// TwinCAT 3 PLC project UnitTestLib
// Title: Unittest
// Company: Hoox.Software
// Author: Patrick Dressel
// ProjectVersion: 0.1
// Description: Basisfunktion zur Erstellung von Unittest und Dokumentation.
// ProgramVersion: 3.1.4022.2
// libraries:
//   Tc2_Standard, * (Beckhoff Automation GmbH)
//   Tc2_System, * (Beckhoff Automation GmbH)
//   Tc2_Utilities, * (Beckhoff Automation GmbH)
//   Base Interfaces,newest,System
// project tree:
//   Datatypes/ EResult_t.TcDUT, EState_t.TcDUT, ObjectId_t.TcDUT (not stored), SResult_t.TcDUT (not stored), SStatistic_t.TcDUT (not stored), StringHandle_t.TcDUT, IdHandle_t.TcDUT, StrMessage_t.TcDUT (not stored), TestCaseHandle_t.TcDUT, TestSuiteHandle_t.TcDUT (not stored)
//   Datatypes/Report/ EExportState_t.TcDUT (not stored), ERetCode_t.TcDUT, NameHandle_t.TcDUT, PathHandle_t.TcDUT, StrFileName_t.TcDUT (not stored), StrPathName_t.TcDUT, UBaseTypes_t.TcDUT (not stored), UTime_t.TcDUT (not stored)
//   Source/ FB_Testsuite.TcPOU, FB_UnitTestBase.TcPOU, PRG_UnitTestLib.TcPOU
//   Source/Report/ FB_TestReportBase.TcPOU, FB_TextReport.TcPOU
//   Version/ Global_Version.TcGVL

// ---- Datatypes/EResult_t.TcDUT
{attribute 'qualified_only'}
{attribute 'strict'}
TYPE EResult_t :
(
	eStatePassed,
	eStateFailed,
	eStateFailedFatal
);
END_TYPE

// ---- Datatypes/EState_t.TcDUT
{attribute 'qualified_only'}
{attribute 'strict'}
TYPE EState_t :
(
	eStateInit,
	eStateIdle,
	eStatePrepare,
	eStateExecute,
	eStateCleanUp,
	eStateReady,
	eStateError
);
END_TYPE

// ---- Datatypes/Report/ERetCode_t.TcDUT
{attribute 'qualified_only'}
{attribute 'strict'}
TYPE ERetCode_t :
(
	eRetFailed := 0,
	eRetBusy,
	eRetDone
);
END_TYPE

// ---- Datatypes/Report/NameHandle_t.TcDUT
TYPE NameHandle_t : Pointer to StrFileName_t; END_TYPE

// ---- Datatypes/Report/PathHandle_t.TcDUT
TYPE PathHandle_t : Pointer to StrFileName_t; END_TYPE

// ---- Datatypes/Report/StrPathName_t.TcDUT
TYPE StrPathName_t : String(255); END_TYPE

// ---- Datatypes/StringHandle_t.TcDUT
TYPE StringHandle_t : POINTER TO STRING(255); END_TYPE

// ---- Datatypes/IdHandle_t.TcDUT
TYPE IdHandle_t : POINTER TO ObjectId_t; END_TYPE

// ---- Datatypes/TestCaseHandle_t.TcDUT
TYPE TestCaseHandle_t : POINTER TO FB_UnitTestBase; END_TYPE

// ---- Version/Global_Version.TcGVL
{attribute 'TcGenerated'}
// This function has been automatically generated from the project information.
VAR_GLOBAL CONSTANT
	{attribute 'const_non_replaced'}
	{attribute 'linkalways'}
	stLibVersion_Unittest : ST_LibVersion := (iMajor := 0, iMinor := 1, iBuild := 0, iRevision := 0, sVersion := '0.1');
END_VAR

// ---- Source/FB_Testsuite.TcPOU
(******************************************************************************
Baustein: FB_Testsuite
Spezifikation: doc/Spezifikation.pdf, Kap. x.y.z
-------------------------------------------------------------------------------
erstellt:
von:
Geändert:
von:
-------------------------------------------------------------------------------
Beschreibung
Dieser Baustein enthält alle zugeordneten Testfälle. Ein Testfall
ist ein abgeleiteter Baustein (FB) von FB_UnitTestBase.

-------------------------------------------------------------------------------
Input
-

Output
-
******************************************************************************)
FUNCTION_BLOCK FB_Testsuite
VAR_INPUT
	i_bStart : BOOL;
END_VAR
VAR_OUTPUT
	o_eState  		: EState_t;
	o_eResult 		: EResult_t;
END_VAR
VAR
	strId			: ObjectId_t;
	bRegistered     : BOOL;
	a_pTest  		: ARRAY [0..255] OF TestCaseHandle_t;
	pTest     		: TestCaseHandle_t;
	u16TestCases  	: UINT;
	u16Index 		: UINT;
	sStatistic 		: SStatistic_t;
END_VAR


	CASE o_eState OF
		
	EState_t.eStateInit:
	
		o_eState 	:= EState_t.eStateError;
		IF bRegistered = TRUE THEN
			o_eState 	:= EState_t.eStateIdle;
		END_IF;
		
	EState_t.eStateIdle:

		u16Index := 0;

		IF i_bStart = TRUE THEN
			logInfo(CONCAT('Run Testsuite ', strId));
			pTest 	 := getFirstTestCase();
			o_eState  := EState_t.eStatePrepare;
			o_eResult := EResult_t.eStatePassed;
		END_IF;

	EState_t.eStatePrepare:
	
		sStatistic.u32Executed  := 0;
		sStatistic.u32Passed 	:= 0;
		sStatistic.u32Failed 	:= 0;
		sStatistic.u32Asserts 	:= 0;

		IF pTest <> 0 THEN
			IF pTest^.prepare() = TRUE THEN
				pTest 	:= getNextTestCase();
			END_IF;
		ELSE
			o_eState := EState_t.eStateExecute;
			pTest 	:= getFirstTestCase();
		END_IF;

	EState_t.eStateExecute:

		IF pTest <> 0 THEN
			IF pTest^.execute() = TRUE THEN

				sStatistic.u32Executed := sStatistic.u32Executed + 1;	
			
				sStatistic.u32Passed 	:= sStatistic.u32Passed + pTest^.getPassed();
				sStatistic.u32Failed 	:= sStatistic.u32Failed + pTest^.getFailed();
				sStatistic.u32Asserts   := sStatistic.u32Passed + sStatistic.u32Failed;
				
				CASE o_eResult OF 

				EResult_t.eStatePassed:
					// Status des letzen Tests übernehmen
					o_eResult := pTest^.o_eResult;

				EResult_t.eStateFailed:
					// Status nur übernehmen wenn ein Fatal-Status
					// ermittelt wird und der Test sofort abgebrochen
					// werden soll.
					IF pTest^.o_eResult = EResult_t.eStateFailedFatal THEN
						o_eResult := pTest^.o_eResult;
						o_eState  := EState_t.eStateCleanUp;
						pTest 	  := getFirstTestCase();	
					END_IF;

				EResult_t.eStateFailedFatal:

					o_eState := EState_t.eStateCleanUp;
					pTest 	:= getFirstTestCase();					

				END_CASE;

				IF o_eResult <> EResult_t.eStateFailedFatal THEN
					pTest 	 := getNextTestCase();
				END_IF;

			END_IF;
		ELSE
			o_eState := EState_t.eStateCleanUp;
			pTest 	:= getFirstTestCase();
		END_IF;

	ESTate_t.eStateCleanUp:

		IF pTest <> 0 THEN
			IF pTest^.cleanup() = TRUE THEN
				pTest 	:= getNextTestCase();
			END_IF;
		ELSE
			o_eState := EState_t.eStateReady;
		END_IF;
		
	ESTate_t.eStateReady:
	
		IF i_bStart = FALSE THEN
			o_eState := EState_t.eStateIdle;
		END_IF
		
	ESTate_t.eStateError:	
		
		// wenn wir hier rauskommen ist was dummes passiert
		
	ELSE
		
		o_eState := EState_t.eStateError;
		
	END_CASE;
	
	
	
	
	
	
//

(******************************************************************************
Baustein: FB_UnitTestBase.
Spezifikation: doc/Spezifikation.pdf, Kap. x.y.z
-------------------------------------------------------------------------------
erstellt:
von:
Geändert:
von:
-------------------------------------------------------------------------------
Beschreibung
Diese Methode

-------------------------------------------------------------------------------
Input
-

Output
-
******************************************************************************)
METHOD PUBLIC addTestcase : BOOL
VAR_INPUT
	i_pTestCase : TestCaseHandle_t;
END_VAR

	addTestcase := FALSE;

	IF 	i_pTestCase  <> 0   AND 
		u16TestCases <  255 THEN
		
		a_pTest[u16TestCases] := i_pTestCase;
		
		u16TestCases := u16TestCases +1;
		
		sStatistic.u32TestCases := sStatistic.u32TestCases + 1;
		
		addTestcase := true;
	END_IF
END_METHOD

METHOD FB_init : BOOL
VAR_INPUT
	bInitRetains 	: BOOL; // if TRUE, the retain variables are initialized (warm start / cold start)
	bInCopyCode 	: BOOL;  // if TRUE, the instance afterwards gets moved into the copy code (online change)
	i_strId	  		: ObjectId_t;
END_VAR

	strId := i_StrId;
	
	register();
END_METHOD

METHOD PUBLIC getExecuted : UDINT
VAR_INPUT
END_VAR

	getExecuted := sStatistic.u32Executed;
END_METHOD

METHOD PUBLIC getFailed : UDINT
VAR_INPUT
END_VAR

	getFailed := sStatistic.u32Failed;
END_METHOD

(******************************************************************************
Baustein: FB_UnitTestBase.
Spezifikation: doc/Spezifikation.pdf, Kap. x.y.z
-------------------------------------------------------------------------------
erstellt:
von:
Geändert:
von:
-------------------------------------------------------------------------------
Beschreibung
Diese Methode

-------------------------------------------------------------------------------
Input
-

Output
-
******************************************************************************)
METHOD PRIVATE getFirstTestCase : TestCaseHandle_t
VAR_INPUT
END_VAR

	u16Index := 0;
	getFirstTestCase := a_pTest[0];
END_METHOD

METHOD PUBLIC getId : STRING
VAR_INPUT
END_VAR

	getId := strId;
END_METHOD

(******************************************************************************
Baustein: FB_UnitTestBase.
Spezifikation: doc/Spezifikation.pdf, Kap. x.y.z
-------------------------------------------------------------------------------
erstellt:
von:
Geändert:
von:
-------------------------------------------------------------------------------
Beschreibung
Diese Methode

-------------------------------------------------------------------------------
Input
-

Output
-
******************************************************************************)
METHOD PRIVATE getNextTestCase : TestCaseHandle_t
VAR_INPUT
END_VAR

	getNextTestCase := 0;
	u16Index 		 := u16Index + 1;

	IF u16Index < u16TestCases THEN
		getNextTestCase := a_pTest[u16Index];
	END_IF;
END_METHOD

METHOD PUBLIC getNoOfAsserts : UDINT
VAR_INPUT
END_VAR

	getNoOfAsserts := sStatistic.u32Asserts;
END_METHOD

METHOD PUBLIC getNoOfTests : UDINT
VAR_INPUT
END_VAR

	getNoOfTests := sStatistic.u32TestCases;
END_METHOD

METHOD PUBLIC getPassed : UDINT
VAR_INPUT
END_VAR

	getPassed := sStatistic.u32Passed;
END_METHOD

METHOD PROTECTED logInfo : BOOL
VAR_INPUT
	i_strMessage : StrMessage_t;
END_VAR

	ADSLOGSTR(msgCtrlMask 	:= ADSLOG_MSGTYPE_HINT , 
			  msgFmtStr 	:= i_strMessage, 
			  strArg 		:= '');
END_METHOD

(******************************************************************************
Baustein: FB_UnitTestBase.
Spezifikation: doc/Spezifikation.pdf, Kap. x.y.z
-------------------------------------------------------------------------------
erstellt:
von:
Geändert:
von:
-------------------------------------------------------------------------------
Beschreibung
Diese Methode

-------------------------------------------------------------------------------
Input
-

Output
-
******************************************************************************)
METHOD PROTECTED register : BOOL
VAR_INPUT
END_VAR

	bRegistered := PRG_UnitTestLib.addTestSuite(this);
END_METHOD

END_FUNCTION_BLOCK

// ---- Source/FB_UnitTestBase.TcPOU
(******************************************************************************
Baustein: FB_UnitTestBase
Spezifikation: doc/Spezifikation.pdf, Kap. x.y.z
-------------------------------------------------------------------------------
erstellt:
von:
Geändert:
von:
-------------------------------------------------------------------------------
Beschreibung
Dieser Baustein stellt die Basis für einen Unittest dar und enthält
alle notwendigen Variablen und Methoden zur Testauswertung.

-------------------------------------------------------------------------------
Input
-

Output
-
******************************************************************************)
FUNCTION_BLOCK FB_UnitTestBase
VAR_INPUT
END_VAR
VAR_OUTPUT
	o_eState : EState_t;
	o_eResult: EResult_t;
END_VAR
VAR
	strId	  		: ObjectId_t;
	pTestSuite      : TestSuiteHandle_t;
	bRegistered 	: BOOL;
	u32Passed 		: UDINT;
	u32Failed 		: UDINT;
END_VAR

(******************************************************************************
Baustein: FB_UnitTestBase.addFailed
Spezifikation: doc/Spezifikation.pdf, Kap. x.y.z
-------------------------------------------------------------------------------
erstellt:
von:
Geändert:
von:
-------------------------------------------------------------------------------
Beschreibung
Diese Methode

-------------------------------------------------------------------------------
Input
-

Output
-
******************************************************************************)
METHOD PRIVATE addFailed : BOOL
VAR_INPUT
	bFatal : BOOL;
END_VAR

	u32Failed := u32Failed + 1;
	
	o_eResult := EResult_t.eStateFailed;
	
	IF bFatal = true THEN
		o_eResult := EResult_t.eStateFailedFatal;
		logError(concat('Test Failed Fatal: ', strId));
	ELSE
		logError(concat('Test Failed : ', strId));
	END_IF
END_METHOD

(******************************************************************************
Baustein: FB_UnitTestBase.
Spezifikation: doc/Spezifikation.pdf, Kap. x.y.z
-------------------------------------------------------------------------------
erstellt:
von:
Geändert:
von:
-------------------------------------------------------------------------------
Beschreibung
Diese Methode

-------------------------------------------------------------------------------
Input
-

Output
-
******************************************************************************)
METHOD PRIVATE addPassed : BOOL
VAR_INPUT
END_VAR

	u32Passed := u32Passed + 1;
END_METHOD

METHOD PROTECTED assertEQUAL : BOOL
VAR_INPUT
	Actual   : ANY;
	Expected : ANY;
END_VAR

	assertEQUAL := FALSE;
	
	IF validate(Actual, Expected) = FALSE THEN
		addFailed(true);
		RETURN;
	END_IF
	
	assertTrue(MEMCMP(Actual.pValue, Expected.pValue, TO_UDINT(Actual.diSize)) = 0);
END_METHOD

METHOD PROTECTED assertEQUAL_Fatal : BOOL
VAR_INPUT
	Actual   : ANY;
	Expected : ANY;
END_VAR

	assertEQUAL_Fatal := FALSE;
	
	IF validate(Actual, Expected) = FALSE THEN
		addFailed(true);
		RETURN;
	END_IF

	assertTrue_Fatal(MEMCMP(Actual.pValue, Expected.pValue, TO_UDINT(Actual.diSize)) = 0);
END_METHOD

(******************************************************************************
Baustein: FB_UnitTestBase.assertFALSE
Spezifikation: doc/Spezifikation.pdf, Kap. x.y.z
-------------------------------------------------------------------------------
erstellt:
von:
Geändert:
von:
-------------------------------------------------------------------------------
Beschreibung
Diese Methode...

-------------------------------------------------------------------------------
Input
-

Output
-
******************************************************************************)
METHOD PROTECTED assertFALSE : BOOL
VAR_INPUT
	bValue : BOOL;
END_VAR

	IF bValue = FALSE THEN
		u32Passed := u32Passed + 1;
	ELSE
		u32Failed := u32Failed + 1;
	END_IF
END_METHOD

(******************************************************************************
Baustein: FB_UnitTestBase.
Spezifikation: doc/Spezifikation.pdf, Kap. x.y.z
-------------------------------------------------------------------------------
erstellt:
von:
Geändert:
von:
-------------------------------------------------------------------------------
Beschreibung
Diese Methode

-------------------------------------------------------------------------------
Input
-

Output
-
******************************************************************************)
METHOD PROTECTED assertFALSE_Fatal : BOOL
VAR_INPUT
	bValue : BOOL;
END_VAR

	IF bValue = FALSE THEN
		addPassed();
	ELSE
		addFailed(bFatal := true);
	END_IF
END_METHOD

METHOD PROTECTED assertNotEqual : BOOL
VAR_INPUT
	Actual   : ANY;
	Expected : ANY;
END_VAR

	assertNotEqual := FALSE;
	
	IF validate(Actual, Expected) = FALSE THEN
		addFailed(true);
		RETURN;
	END_IF
	
	assertTrue(MEMCMP(Actual.pValue, Expected.pValue, TO_UDINT(Actual.diSize)) <> 0);
END_METHOD

METHOD PROTECTED assertNotEqual_Fatal : BOOL
VAR_INPUT
	Actual   : ANY;
	Expected : ANY;
END_VAR

	assertNotEqual_Fatal := FALSE;
	
	IF validate(Actual, Expected) = FALSE THEN
		addFailed(true);
		RETURN;
	END_IF
	
	assertTrue_Fatal(MEMCMP(Actual.pValue, Expected.pValue, TO_UDINT(Actual.diSize)) <> 0);
END_METHOD

(******************************************************************************
Baustein: FB_UnitTestBase.
Spezifikation: doc/Spezifikation.pdf, Kap. x.y.z
-------------------------------------------------------------------------------
erstellt:
von:
Geändert:
von:
-------------------------------------------------------------------------------
Beschreibung
Diese Methode

-------------------------------------------------------------------------------
Input
-

Output
-
******************************************************************************)
METHOD PROTECTED assertPtrEqual : BOOL
VAR_INPUT
	pActual   : PVOID;
	pExpected : PVOID;
END_VAR

	assertTRUE(pActual = pExpected);
END_METHOD

(******************************************************************************
Baustein: FB_UnitTestBase.
Spezifikation: doc/Spezifikation.pdf, Kap. x.y.z
-------------------------------------------------------------------------------
erstellt:
von:
Geändert:
von:
-------------------------------------------------------------------------------
Beschreibung
Diese Methode

-------------------------------------------------------------------------------
Input
-

Output
-
******************************************************************************)
METHOD PROTECTED assertPtrEqual_Fatal : BOOL
VAR_INPUT
	pActual   : PVOID;
	pExpected : PVOID;
END_VAR

	assertTRUE_Fatal(pActual = pExpected);
END_METHOD

(******************************************************************************
Baustein: FB_UnitTestBase.
Spezifikation: doc/Spezifikation.pdf, Kap. x.y.z
-------------------------------------------------------------------------------
erstellt:
von:
Geändert:
von:
-------------------------------------------------------------------------------
Beschreibung
Diese Methode

-------------------------------------------------------------------------------
Input
-

Output
-
******************************************************************************)
METHOD PROTECTED assertPtrNotEqual : BOOL
VAR_INPUT
	pActual   : PVOID;
	pExpected : PVOID;
END_VAR

	assertTRUE(pActual <> pExpected);
END_METHOD

(******************************************************************************
Baustein: FB_UnitTestBase.
Spezifikation: doc/Spezifikation.pdf, Kap. x.y.z
-------------------------------------------------------------------------------
erstellt:
von:
Geändert:
von:
-------------------------------------------------------------------------------
Beschreibung
Diese Methode

-------------------------------------------------------------------------------
Input
-

Output
-
******************************************************************************)
METHOD PROTECTED assertPtrNotEqual_Fatal : BOOL
VAR_INPUT
	pActual   : PVOID;
	pExpected : PVOID;
END_VAR

	assertTRUE_Fatal(pActual <> pExpected);
END_METHOD

(******************************************************************************
Baustein: FB_UnitTestBase.
Spezifikation: doc/Spezifikation.pdf, Kap. x.y.z
-------------------------------------------------------------------------------
erstellt:
von:
Geändert:
von:
-------------------------------------------------------------------------------
Beschreibung
Diese Methode

-------------------------------------------------------------------------------
Input
-

Output
-
******************************************************************************)
METHOD PROTECTED assertPtrNotNull : BOOL
VAR_INPUT
	pActual   : PVOID;
END_VAR

	assertTRUE(pActual <> 0);
END_METHOD

(******************************************************************************
Baustein: FB_UnitTestBase.
Spezifikation: doc/Spezifikation.pdf, Kap. x.y.z
-------------------------------------------------------------------------------
erstellt:
von:
Geändert:
von:
-------------------------------------------------------------------------------
Beschreibung
Diese Methode

-------------------------------------------------------------------------------
Input
-

Output
-
******************************************************************************)
METHOD PROTECTED assertPtrNotNull_Fatal : BOOL
VAR_INPUT
	pActual   : PVOID;
END_VAR

	assertTRUE_Fatal(pActual <> 0);
END_METHOD

(******************************************************************************
Baustein: FB_UnitTestBase.
Spezifikation: doc/Spezifikation.pdf, Kap. x.y.z
-------------------------------------------------------------------------------
erstellt:
von:
Geändert:
von:
-------------------------------------------------------------------------------
Beschreibung
Diese Methode

-------------------------------------------------------------------------------
Input
-

Output
-
******************************************************************************)
METHOD PROTECTED assertPtrNull : BOOL
VAR_INPUT
	pActual   : PVOID;
END_VAR

	assertTRUE(pActual = 0);
END_METHOD

(******************************************************************************
Baustein: FB_UnitTestBase.
Spezifikation: doc/Spezifikation.pdf, Kap. x.y.z
-------------------------------------------------------------------------------
erstellt:
von:
Geändert:
von:
-------------------------------------------------------------------------------
Beschreibung
Diese Methode

-------------------------------------------------------------------------------
Input
-

Output
-
******************************************************************************)
METHOD PROTECTED assertPtrNull_Fatal : BOOL
VAR_INPUT
	pActual   : PVOID;
END_VAR

	assertTRUE_Fatal(pActual = 0);
END_METHOD

(******************************************************************************
Baustein: FB_UnitTestBase.
Spezifikation: doc/Spezifikation.pdf, Kap. x.y.z
-------------------------------------------------------------------------------
erstellt:
von:
Geändert:
von:
-------------------------------------------------------------------------------
Beschreibung
Diese Methode

-------------------------------------------------------------------------------
Input
-

Output
-
******************************************************************************)
METHOD PROTECTED assertRealEqual : BOOL
VAR_INPUT
	r32Actual 		: REAL;
	r32Expected 	: REAL;
	r32Granularity 	: REAL;
END_VAR

	assertTRUE(ABS(r32Actual-r32Expected) <= ABS(r32Granularity));
END_METHOD

(******************************************************************************
Baustein: FB_UnitTestBase.
Spezifikation: doc/Spezifikation.pdf, Kap. x.y.z
-------------------------------------------------------------------------------
erstellt:
von:
Geändert:
von:
-------------------------------------------------------------------------------
Beschreibung
Diese Methode

-------------------------------------------------------------------------------
Input
-

Output
-
******************************************************************************)
METHOD PROTECTED assertRealEqual_Fatal : BOOL
VAR_INPUT
	r32Actual 		: REAL;
	r32Expected 	: REAL;
	r32Granularity 	: REAL;
END_VAR

	assertTRUE_Fatal(ABS(r32Actual-r32Expected) <= ABS(r32Granularity));
END_METHOD

(******************************************************************************
Baustein: FB_UnitTestBase.
Spezifikation: doc/Spezifikation.pdf, Kap. x.y.z
-------------------------------------------------------------------------------
erstellt:
von:
Geändert:
von:
-------------------------------------------------------------------------------
Beschreibung
Diese Methode

-------------------------------------------------------------------------------
Input
-

Output
-
******************************************************************************)
METHOD PRIVATE assertRealNotEqual : BOOL
VAR_INPUT
	r32Actual 		: REAL;
	r32Expected 	: REAL;
	r32Granularity 	: REAL;
END_VAR

	assertTRUE(ABS(r32Actual-r32Expected) > ABS(r32Granularity));
END_METHOD

(******************************************************************************
Baustein: FB_UnitTestBase.
Spezifikation: doc/Spezifikation.pdf, Kap. x.y.z
-------------------------------------------------------------------------------
erstellt:
von:
Geändert:
von:
-------------------------------------------------------------------------------
Beschreibung
Diese Methode

-------------------------------------------------------------------------------
Input
-

Output
-
******************************************************************************)
METHOD PROTECTED assertRealNotEqual_Fatal : BOOL
VAR_INPUT
	r32Actual 		: REAL;
	r32Expected 	: REAL;
	r32Granularity 	: REAL;
END_VAR

	assertTRUE_Fatal(ABS(r32Actual-r32Expected) > ABS(r32Granularity));
END_METHOD

(******************************************************************************
Baustein: FB_UnitTestBase.
Spezifikation: doc/Spezifikation.pdf, Kap. x.y.z
-------------------------------------------------------------------------------
erstellt:
von:
Geändert:
von:
-------------------------------------------------------------------------------
Beschreibung
Diese Methode

-------------------------------------------------------------------------------
Input
-

Output
-
******************************************************************************)
METHOD PROTECTED assertStringEqual : BOOL
VAR_INPUT
	pActual 	: StringHandle_t;
	pExpected 	: StringHandle_t;
END_VAR

	IF strncmp(pActual, pExpected, LEN(pExpected^)) = TRUE THEN
		addPassed();
	ELSE
		addFailed(bFatal := FALSE);		
	END_IF
END_METHOD

(******************************************************************************
Baustein: FB_UnitTestBase.
Spezifikation: doc/Spezifikation.pdf, Kap. x.y.z
-------------------------------------------------------------------------------
erstellt:
von:
Geändert:
von:
-------------------------------------------------------------------------------
Beschreibung
Diese Methode

-------------------------------------------------------------------------------
Input
-

Output
-
******************************************************************************)
METHOD PROTECTED assertStringEqual_Fatal : BOOL
VAR_INPUT
	pActual 	: StringHandle_t;
	pExpected 	: StringHandle_t;
END_VAR

	IF strncmp(pActual, pExpected, LEN(pExpected^)) = TRUE THEN
		addPassed();
	ELSE
		addFailed(bFatal := TRUE);		
	END_IF
END_METHOD

(******************************************************************************
Baustein: FB_UnitTestBase.
Spezifikation: doc/Spezifikation.pdf, Kap. x.y.z
-------------------------------------------------------------------------------
erstellt:
von:
Geändert:
von:
-------------------------------------------------------------------------------
Beschreibung
Diese Methode

-------------------------------------------------------------------------------
Input
-

Output
-
******************************************************************************)
METHOD PROTECTED assertStringNotEqual : BOOL
VAR_INPUT
	pActual 	: StringHandle_t;
	pExpected 	: StringHandle_t;
END_VAR

	IF strncmp(pActual, pExpected, LEN(pExpected^)) = false THEN
		addPassed();
	ELSE
		addFailed(bFatal := FALSE);		
	END_IF
END_METHOD

(******************************************************************************
Baustein: FB_UnitTestBase.
Spezifikation: doc/Spezifikation.pdf, Kap. x.y.z
-------------------------------------------------------------------------------
erstellt:
von:
Geändert:
von:
-------------------------------------------------------------------------------
Beschreibung
Diese Methode

-------------------------------------------------------------------------------
Input
-

Output
-
******************************************************************************)
METHOD PROTECTED assertStringNotEqual_fatal : BOOL
VAR_INPUT
	pExpected 	: StringHandle_t;
	pActual 	: StringHandle_t;
END_VAR

	IF strncmp(pActual, pExpected, LEN(pExpected^)) = FALSE THEN
		addPassed();
	ELSE
		addFailed(bFatal := TRUE);		
	END_IF
END_METHOD

(******************************************************************************
Baustein: FB_UnitTestBase.assertTRUE
Spezifikation: doc/Spezifikation.pdf, Kap. x.y.z
-------------------------------------------------------------------------------
erstellt:
von:
Geändert:
von:
-------------------------------------------------------------------------------
Beschreibung
Diese Methode...

-------------------------------------------------------------------------------
Input
-

Output
-
******************************************************************************)
METHOD PROTECTED assertTRUE : BOOL
VAR_INPUT
	bValue : BOOL;
END_VAR

	IF bValue = true THEN
		addPassed();
	ELSE
		addFailed(bFatal := FALSE);
	END_IF
END_METHOD


(******************************************************************************
Baustein: FB_UnitTestBase.
Spezifikation: doc/Spezifikation.pdf, Kap. x.y.z
-------------------------------------------------------------------------------
erstellt:
von:
Geändert:
von:
-------------------------------------------------------------------------------
Beschreibung
Diese Methode

-------------------------------------------------------------------------------
Input
-

Output
-
******************************************************************************)
METHOD PROTECTED assertTRUE_Fatal : BOOL
VAR_INPUT
	bValue : BOOL;
END_VAR

	IF bValue = TRUE THEN
		addPassed();
	ELSE
		addFailed(bFatal := true);
	END_IF
END_METHOD

(******************************************************************************
Baustein: FB_UnitTestBase.cleanup
Spezifikation: doc/Spezifikation.pdf, Kap. x.y.z
-------------------------------------------------------------------------------
erstellt:
von:
Geändert:
von:
-------------------------------------------------------------------------------
Beschreibung
Diese Methode...

-------------------------------------------------------------------------------
Input
-

Output
-
******************************************************************************)
METHOD PUBLIC cleanup : BOOL
VAR_INPUT
END_VAR

	cleanup := TRUE;
END_METHOD

(******************************************************************************
Baustein: FB_UnitTestBase.execute
Spezifikation: doc/Spezifikation.pdf, Kap. x.y.z
-------------------------------------------------------------------------------
erstellt:
von:
Geändert:
von:
-------------------------------------------------------------------------------
Beschreibung
Diese Methode...

-------------------------------------------------------------------------------
Input
-

Output
-
******************************************************************************)
METHOD PUBLIC execute : BOOL
VAR_INPUT
END_VAR

	Execute := TRUE;
END_METHOD

METHOD FB_init : BOOL
VAR_INPUT
	bInitRetains 	: BOOL; // if TRUE, the retain variables are initialized (warm start / cold start)
	bInCopyCode 	: BOOL;  // if TRUE, the instance afterwards gets moved into the copy code (online change)
	i_strId	  		: ObjectId_t;
	i_pTestSuite 	: TestSuiteHandle_t;
	i_bExecute      : BOOL := true; 
END_VAR
	
	strId 		:= i_strId;
	pTestSuite 	:= i_pTestSuite;
	
	register();
END_METHOD

METHOD PUBLIC getFailed : UDINT
VAR_INPUT
END_VAR

	getFailed := u32Failed;
END_METHOD

METHOD PUBLIC getPassed : UDINT
VAR_INPUT
END_VAR

	getPassed := u32Passed;
END_METHOD

METHOD PROTECTED logError : BOOL
VAR_INPUT
	i_strMessage : StrMessage_t;
END_VAR

	ADSLOGSTR(msgCtrlMask 	:= ADSLOG_MSGTYPE_ERROR , 
			  msgFmtStr 	:= i_strMessage, 
			  strArg 		:= '');
END_METHOD

METHOD PROTECTED logInfo : BOOL
VAR_INPUT
	i_strMessage : StrMessage_t;
END_VAR

	ADSLOGSTR(msgCtrlMask 	:= ADSLOG_MSGTYPE_HINT , 
			  msgFmtStr 	:= i_strMessage, 
			  strArg 		:= '');
END_METHOD

(******************************************************************************
Baustein: FB_UnitTestBase.prepare
Spezifikation: doc/Spezifikation.pdf, Kap. x.y.z
-------------------------------------------------------------------------------
erstellt:
von:
Geändert:
von:
-------------------------------------------------------------------------------
Beschreibung
Diese Methode...

-------------------------------------------------------------------------------
Input
-

Output
-
******************************************************************************)
METHOD PUBLIC prepare : BOOL
VAR_INPUT
END_VAR

	u32Passed := 0;
	u32Failed := 0;
	
	prepare := true;
END_METHOD

(******************************************************************************
Baustein: FB_UnitTestBase.
Spezifikation: doc/Spezifikation.pdf, Kap. x.y.z
-------------------------------------------------------------------------------
erstellt:
von:
Geändert:
von:
-------------------------------------------------------------------------------
Beschreibung
Diese Methode

-------------------------------------------------------------------------------
Input
-

Output
-
******************************************************************************)
METHOD PROTECTED register : BOOL
VAR_INPUT
END_VAR

	IF pTestSuite <> 0 	AND 
       bRegistered = FALSE  THEN
		
		bRegistered := pTestSuite^.addTestcase(THIS);
	
	END_IF
END_METHOD

(******************************************************************************
Baustein: FB_UnitTestBase.
Spezifikation: doc/Spezifikation.pdf, Kap. x.y.z
-------------------------------------------------------------------------------
erstellt:
von:
Geändert:
von:
-------------------------------------------------------------------------------
Beschreibung
Diese Methode

-------------------------------------------------------------------------------
Input
-

Output
-
******************************************************************************)
METHOD PRIVATE strncmp : BOOL
VAR_INPUT
	strInput 	: StringHandle_t;
	strCompare 	: StringHandle_t;
	s16Size		: INT;
END_VAR
VAR
	s16Size1 : INT;
	s16Size2 : INT;
	s16Diff  : INT;
END_VAR

   s16Size1:= LEN(strInput^); 
	s16Size2:= LEN(strCompare^); 
	
	strncmp := FALSE;
	
	s16Diff := s16Size1 - s16Size2;
   
	// vergleich nur wenn beide Strings
	// gleich groß sind.
	IF s16Diff  = 0 THEN

		strncmp := TRUE;
	
		WHILE(s16Size > 0) DO

			IF strInput^ <> strCompare^ THEN
				strncmp := FALSE;
			END_IF;  
 
			strInput   := strInput + 1;
			strCompare := strCompare + 1;
			s16Size    := s16Size - 1;

		END_WHILE


	
	END_IF;
END_METHOD

METHOD PRIVATE validate : BOOL
VAR_INPUT
	var1 : ANY;
	var2 : ANY;
END_VAR

	validate := FALSE;
	
	IF (var1.pValue = 0 OR var1.pValue = 0) THEN
		RETURN;
	END_IF

	IF (var1.TypeClass <> var1.TypeClass) THEN
		RETURN;
	END_IF;	
	
	IF (var1.diSize <> var1.diSize) THEN
		RETURN;
	END_IF;	
	
	validate := true;
END_METHOD

END_FUNCTION_BLOCK

// ---- Source/PRG_UnitTestLib.TcPOU
(******************************************************************************
Baustein: PRG_TestLibrary
Spezifikation: doc/Spezifikation.pdf, Kap. x.y.z
-------------------------------------------------------------------------------
erstellt:
von:
Geändert:
von:
-------------------------------------------------------------------------------
Beschreibung
Dieser Baustein etnhält alle Testsuites und führt diese aus.

-------------------------------------------------------------------------------
Input
-

Output
-
******************************************************************************)
{attribute 'global_init_slot' := '41000'}
PROGRAM PRG_UnitTestLib
VAR_INPUT
	i_bStart : BOOL;
END_VAR
VAR_OUTPUT
	o_eState  		: EState_t;
	o_eResult 		: EResult_t;
	o_sStatistic	: SStatistic_t;
END_VAR
VAR
	a_pTestSuite 	: ARRAY [0..255] OF TestSuiteHandle_t;
	u16TestSuites 	: UINT;
	u16Index	  	: UINT;
	pActTestSuite 	: TestSuiteHandle_t;
	pTestReport		: POINTER TO FB_TestReportBase;
	eRetCode 		: ERetCode_t;

	fbSystemTime 	: FB_LocalSystemTime;
END_VAR


	fbSystemTime(bEnable := true, dwCycle := 5);

	CASE o_eState OF 
	
	EState_t.eStateInit:	
	
		IF i_bStart = FALSE THEN
			o_eState := EState_t.eStateIdle;
		END_IF
	
	EState_t.eStateIdle:
	
		IF i_bStart = TRUE THEN
			logInfo('+++++++++++++ Testbeginn ++++++++++++++');
			o_eState := EState_t.eStatePrepare;
		END_IF
	
	EState_t.eStatePrepare:
	
		o_eResult 	  				:= EResult_t.eStatePassed;
		o_sStatistic.u32Executed 	:= 0;
		o_sStatistic.u32TestCases	:= 0;
		o_sStatistic.u32Asserts  	:= 0;
		o_sStatistic.u32Passed   	:= 0;
		o_sStatistic.u32Failed	 	:= 0;		
		pActTestSuite := getFirstTestSuite();
		
		IF pActTestSuite <> 0 THEN
			o_eState := EState_t.eStateExecute;
		ELSE
			o_eState := EState_t.eStateError;	
		END_IF
	
	EState_t.eStateExecute:
	
		pActTestSuite^(i_bStart := TRUE);
	
		IF pActTestSuite^.o_eState = EState_t.eStateReady THEN
			
			IF pActTestSuite^.o_eResult = EResult_t.eStateFailed THEN
				o_eResult := EResult_t.eStateFailed;
			END_IF
			
			pActTestSuite^(i_bStart := FALSE);
			
			o_eState := EState_t.eStateCleanUp;
			
			o_sStatistic.u32Executed 	:= o_sStatistic.u32Executed  + pActTestSuite^.getExecuted();
			o_sStatistic.u32TestCases	:= o_sStatistic.u32TestCases + pActTestSuite^.getNoOfTests(); 
			o_sStatistic.u32Asserts  	:= o_sStatistic.u32Asserts   + pActTestSuite^.getNoOfAsserts();
			o_sStatistic.u32Passed   	:= o_sStatistic.u32Passed    + pActTestSuite^.getPassed();
			o_sStatistic.u32Failed	 	:= o_sStatistic.u32Failed    + pActTestSuite^.getFailed();
		END_IF
	
	EState_t.eStateCleanUp:
	
		IF pActTestSuite^.o_eResult = EResult_t.eStateFailedFatal THEN
			o_eResult := EResult_t.eStateFailedFatal;
			o_eState  := EState_t.eStateReady;
		ELSE
			
			pActTestSuite := getNextTestSuite();
						
			IF pActTestSuite <> 0 THEN
				o_eState := EState_t.eStateExecute;
			ELSE
				o_eState := EState_t.eStateReady;
				logInfo('+++++++++++++ Test Ende ++++++++++++++');
			END_IF		
			
		END_IF
		
	EState_t.eStateReady:

		IF i_bStart = FALSE THEN
			o_eState := EState_t.eStateExport;
		END_IF

	EState_t.eStateExport:

		IF pTestReport <> 0 THEN
			eRetCode := pTestReport^.create();
		ELSE
			o_eState := EState_t.eStateError;
		END_IF;

		IF eRetCode = ERetCode_t.eRetDone THEN
			o_eState := EState_t.eStateIdle;
		END_IF;

		IF eRetCode = ERetCode_t.eRetFailed THEN
			o_eState := EState_t.eStateError;
		END_IF;

	EState_t.eStateError:
	
	END_CASE

METHOD PUBLIC addTestReport : BOOL
VAR_INPUT
	i_pTestReport : Pointer to FB_TestReportBase;
END_VAR

	pTestReport := i_pTestReport;
END_METHOD

(******************************************************************************
Baustein: FB_UnitTestBase.
Spezifikation: doc/Spezifikation.pdf, Kap. x.y.z
-------------------------------------------------------------------------------
erstellt:
von:
Geändert:
von:
-------------------------------------------------------------------------------
Beschreibung
Diese Methode

-------------------------------------------------------------------------------
Input
-

Output
-
******************************************************************************)
METHOD PUBLIC addTestSuite : BOOL
VAR_INPUT
	i_pTestSuite : TestSuiteHandle_t;
END_VAR

	addTestSuite := FALSE;

	IF 	i_pTestSuite  <> 0   AND 
		u16TestSuites <  255 THEN
		
		a_pTestSuite[u16TestSuites] := i_pTestSuite;
		
		u16TestSuites := u16TestSuites +1;
	
		o_sStatistic.u32TestSuites := o_sStatistic.u32TestSuites + 1;
		o_sStatistic.u32TestCases  := o_sStatistic.u32TestCases + i_pTestSuite^.sStatistic.u32TestCases;
		
		addTestSuite := TRUE;
	END_IF
END_METHOD

(******************************************************************************
Baustein: FB_UnitTestBase.
Spezifikation: doc/Spezifikation.pdf, Kap. x.y.z
-------------------------------------------------------------------------------
erstellt:
von:
Geändert:
von:
-------------------------------------------------------------------------------
Beschreibung
Diese Methode

-------------------------------------------------------------------------------
Input
-

Output
-
******************************************************************************)
METHOD PRIVATE getFirstTestSuite : TestSuiteHandle_t
VAR_INPUT
END_VAR

	u16Index := 0;
	getFirstTestSuite := a_pTestSuite[0];
END_METHOD

(******************************************************************************
Baustein: FB_UnitTestBase.
Spezifikation: doc/Spezifikation.pdf, Kap. x.y.z
-------------------------------------------------------------------------------
erstellt:
von:
Geändert:
von:
-------------------------------------------------------------------------------
Beschreibung
Diese Methode

-------------------------------------------------------------------------------
Input
-

Output
-
******************************************************************************)
METHOD PRIVATE getNextTestSuite : TestSuiteHandle_t
VAR_INPUT
END_VAR

	getNextTestSuite := 0;
	u16Index 		 := u16Index + 1;

	IF u16Index < u16TestSuites THEN
		getNextTestSuite := a_pTestSuite[u16Index];
	END_IF;
END_METHOD

METHOD getTime : TimeStruct
VAR_INPUT
END_VAR
VAR
END_VAR

	getTime := fbSystemTime.systemTime;
END_METHOD

METHOD PROTECTED logInfo : BOOL
VAR_INPUT
	i_strMessage : StrMessage_t;
END_VAR

	ADSLOGSTR(msgCtrlMask 	:= ADSLOG_MSGTYPE_HINT , 
			  msgFmtStr 	:= i_strMessage, 
			  strArg 		:= '');
END_METHOD

END_PROGRAM

// ---- Source/Report/FB_TestReportBase.TcPOU
(******************************************************************************
Baustein: FB_TestReportBase
Spezifikation: doc/Spezifikation.pdf, Kap. x.y.z
-------------------------------------------------------------------------------
erstellt:
von:
Geändert:
von:
-------------------------------------------------------------------------------
Beschreibung
Dieser Baustein enthält alle zugeordneten Testfälle. Ein Testfall
ist ein abgeleiteter Baustein (FB) von FB_UnitTestBase.

-------------------------------------------------------------------------------
Input
-

Output
-
******************************************************************************)
FUNCTION_BLOCK FB_TestReportBase
VAR_INPUT
END_VAR
VAR_OUTPUT
END_VAR
VAR
	strBuffer   : STRING(255);
	fbOpen      : FB_FileOpen;
	fbClose     : FB_FileClose;
	fbWrite	    : FB_FileWrite;
	strFileName : StrFileName_t;
	strFilePath : StrPathName_t;
	
	eState 		: EExportState_t;
	u32Line     : UDINT;
	
	sStatistic  : SStatistic_t;

	trgOpen 	: F_TRIG;
	trgWrite 	: F_TRIG;
	trgClose 	: F_TRIG;
END_VAR

METHOD PROTECTED addCrlf : BOOL
VAR_INPUT
END_VAR
VAR
END_VAR
   
	strBuffer := CONCAT(strBuffer, '$R$N');
END_METHOD

METHOD PROTECTED addDate : ERetCode_t
VAR_INPUT
	i_sDate : TIMESTRUCT;
END_VAR

   	addDate := ERetcode_t.eRetDone;

   	addValue(i_sDate.wDay);
   	addString('.');
   	addValue(i_sDate.wMonth);
   	addString('.');
    addValue(i_sDate.wYear);
    addString(' ');
END_METHOD

METHOD PROTECTED addString : ERetCode_t
VAR_INPUT
	i_strData : STRING(255);
END_VAR

	strBuffer :=  concat(strBuffer, i_strData);

	addString := ERetcode_t.eRetDone;
END_METHOD

METHOD PROTECTED addTime : ERetCode_t
VAR_INPUT
	i_sTime : TIMESTRUCT;
END_VAR

	addTime := ERetcode_t.eRetDone;
	
   	addValue(i_sTime.wHour);
   	addString('.');
   	addValue(i_sTime.wMinute);
  	addString('.');
   	addValue(i_sTime.wSecond);
   	addString(' ');
END_METHOD

METHOD PROTECTED addValue : ERetCode_t
VAR_INPUT
	i_anyValue : ANY;
END_VAR
VAR
	uValue : UBaseTypes_t;
END_VAR

	addValue  := ERetcode_t.eRetDone;
	
	IF i_anyValue.pValue = 0 THEN
		addValue  := ERetcode_t.eRetFailed;
		RETURN;
	END_IF

	MEMCPY(ADR(uValue),i_anyValue.pValue, TO_UDINT(i_anyValue.diSize)); 

	CASE i_anyValue.TypeClass OF

	IBaseLibrary.TYPE_SINT:

		addString(SINT_TO_STRING(uValue.s8Value));

	//IBaseLibrary.TYPE_BYTE:
	IBaseLibrary.TYPE_USINT:

		addString(USINT_TO_STRING(uValue.u8Value));

	IBaseLibrary.TYPE_INT:

		addString(INT_TO_STRING(uValue.s16Value));

	IBaseLibrary.TYPE_DINT:

		addString(DINT_TO_STRING(uValue.s32Value));

	IBaseLibrary.TYPE_UINT:

		addString(UINT_TO_STRING(uValue.u16Value));

	IBaseLibrary.TYPE_UDINT:

		addString(UDINT_TO_STRING(uValue.u32Value));

	IBaseLibrary.TYPE_WORD:

		addString(WORD_TO_STRING(uValue.w16Value));

	IBaseLibrary.TYPE_DWORD:

		addString(DWORD_TO_STRING(uValue.w32Value));

	ELSE
		ADSLOGSTR(msgCtrlMask 	:= ADSLOG_MSGTYPE_ERROR , 
				  msgFmtStr 	:= 'TestReportBase.AddValue: Unbekannter Datentyp!', 
				  strArg 		:= '');
	END_CASE;
END_METHOD

(******************************************************************************
Baustein: FB_TestReportBase.BuildFile
Spezifikation: doc/Spezifikation.pdf, Kap. x.y.z
-------------------------------------------------------------------------------
erstellt:
von:
Geändert:
von:
-------------------------------------------------------------------------------
Beschreibung
Diese Methode muss vom ableitenden Baustein überschrieben werden und
wird von der Basisklasse aus aufgerufen wenn der Report erstellt werden
soll.

-------------------------------------------------------------------------------
Input
-

Output
-
******************************************************************************)
METHOD PROTECTED BuildFile : ERetCode_t
VAR_INPUT
	i_u32Line : UDINT;
END_VAR
END_METHOD

METHOD PROTECTED clearBuffer : ERetCode_t
VAR_INPUT
END_VAR

	clearBuffer := ERetCode_t.eRetDone;
	
	strBuffer := '';
END_METHOD

METHOD PROTECTED Close : ERetCode_t
VAR_INPUT
END_VAR

	Close := ERetCode_t.eRetFailed;
	
	fbClose.hFile 		:= fbOpen.hFile;
	fbClose.bExecute 	:= TRUE; 

	IF trgClose.Q = TRUE THEN
		Close := ERetCode_t.eRetDone;
		fbClose.bExecute  := FALSE;		
	ELSE	
		Close := ERetCode_t.eRetBusy;
	END_IF;	
	
	IF fbClose.bError = TRUE THEN
		Close := eRetCode_t.eRetFailed;
	END_IF;
END_METHOD

METHOD PUBLIC create : ERetCode_t;
VAR_INPUT
END_VAR
VAR
	eRetCode : ERetCode_t;
END_VAR

	create := ERetCode_t.eRetBusy;

	fbOpen();
	fbWrite();
	fbClose();

	trgOpen(CLK := fbOpen.bBusy);
	trgWrite(CLK := fbWrite.bBusy);
	trgClose(CLK := fbClose.bBusy);
	
	CASE eState OF
	
	EExportState_t.eExportIdle:
	
		eState := EExportState_t.eExportOpen;
	
	EExportState_t.eExportOpen:
	
		eRetCode 	:= Open();
		u32Line  	:= 0;
		sStatistic 	:= PRG_UnitTestLib.o_sStatistic;

		IF eRetCode = ERetCode_t.eRetDone THEN
			eState := EExportState_t.eExportGetLine;
		ELSIF eRetCode = ERetCode_t.eRetFailed THEN
			eState := EExportState_t.eExportError;
		END_IF;

	EExportState_t.eExportGetLine:

		eRetCode := BuildFile(u32Line);

		IF eRetCode = ERetCode_t.eRetDone THEN
			eState := EExportState_t.eExportClose;
		ELSIF eRetCode = ERetCode_t.eRetFailed THEN
			eState := EExportState_t.eExportError;
		ELSE
			addCrlf();
			eState := EExportState_t.eExportWrite;
		END_IF;

	EExportState_t.eExportWrite:
	
		IF writeBuffer() =  ERetCode_t.eRetDone THEN
			clearBuffer();	
			u32Line := u32Line + 1;
			eState  := EExportState_t.eExportGetLine;
		END_IF;		
	
	EExportState_t.eExportClose:
	
		eRetCode := Close();
		
		IF eRetCode = ERetCode_t.eRetDone THEN
			eState     := EExportState_t.eExportIdle;
			create	   := ERetCode_t.eRetDone;
			reset();
		ELSIF eRetCode = ERetCode_t.eRetFailed THEN
			eState := EExportState_t.eExportError;
		end_if;
	
	EExportState_t.eExportError:
	
		create := ERetCode_t.eRetFailed;
	
	end_case;
END_METHOD

(******************************************************************************
Baustein: FB_TestReportBase.getFileName
Spezifikation: doc/Spezifikation.pdf, Kap. x.y.z
-------------------------------------------------------------------------------
erstellt:
von:
Geändert:
von:
-------------------------------------------------------------------------------
Beschreibung
Diese Methode muss vom ableitenden Baustein überschrieben werden und
wird von der Basisklasse aus aufgerufen wenn der Report erstellt werden
soll.

-------------------------------------------------------------------------------
Input
-

Output
-
******************************************************************************)
METHOD PROTECTED getFileName : ERetCode_t
VAR_INPUT
	i_pFileName : NameHandle_t;
	i_pPath		: PathHandle_t;
END_VAR
END_METHOD

METHOD PROTECTED getTime : TimeStruct
VAR_INPUT
END_VAR
VAR
END_VAR

	getTime := PRG_UnitTestLib.getTime();
END_METHOD

METHOD PROTECTED open : ERetCode_t
VAR_INPUT
END_VAR

	open := ERetCode_t.eRetFailed;

	getFileName(ADR(strFileName), ADR(strFilePath));
	
	fbOpen.sPathName := CONCAT(strFilePath, strFileName);
	fbOpen.nMode 	 := FOPEN_MODEWRITE OR FOPEN_MODEBINARY;	
	fbOpen.bExecute  := TRUE;
			
	IF trgOpen.Q = TRUE THEN
		open := ERetCode_t.eRetDone;
		fbOpen.bExecute  := FALSE;		
	ELSE	
		open := ERetCode_t.eRetBusy;
	END_IF;	
	
	IF fbOpen.bError = TRUE THEN
		open := eRetCode_t.eRetFailed;
	END_IF;
END_METHOD

METHOD PUBLIC reset : BOOL
VAR_INPUT
END_VAR

	IF fbOpen.hFile <> 0 THEN
		close();
	END_IF
	
	clearBuffer();

	fbOpen(sPathName := '', bExecute := FALSE);
	
	fbWrite(bExecute := FALSE);
	
	fbClose(bExecute := FALSE);
	
	eState := EExportState_t.eExportIdle;
END_METHOD

METHOD PROTECTED writeBuffer : ERetCode_t
VAR_INPUT
END_VAR
VAR
	u32Len : UDINT;
END_VAR

	writeBuffer := eRetCode_t.eRetBusy;
	
	IF LEN(strBuffer) <= 0 THEN
		RETURN;
	END_IF
	
	u32Len := TO_UDINT(LEN(strBuffer)); 
	
	writeBuffer := writeData(i_pData := ADR(strBuffer), u32Size := u32Len);
END_METHOD

METHOD PROTECTED writeData : ERetCode_t
VAR_INPUT
	i_pData : POINTER TO BYTE;
	u32Size : UDINT;
END_VAR

	writeData := ERetCode_t.eRetFailed;
	
	IF u32Size = 0 OR i_pData = 0 THEN
		RETURN;
	END_IF
	
	fbWrite.pWriteBuff 	:= i_pData; 
	fbWrite.cbWriteLen 	:= u32Size; 
	fbWrite.hFile 		:= fbOpen.hFile; 
	fbWrite.bExecute 	:= TRUE;
			
	IF trgWrite.Q = TRUE THEN
		writeData := ERetCode_t.eRetDone;
		fbWrite.bExecute 	:= FALSE;			
	ELSE	
		writeData := ERetCode_t.eRetBusy;
	END_IF;	

	IF fbWrite.bError = TRUE THEN
		writeData := eRetCode_t.eRetFailed;
	END_IF;
END_METHOD

END_FUNCTION_BLOCK

// ---- Source/Report/FB_TextReport.TcPOU
FUNCTION_BLOCK FB_TextReport EXTENDS FB_TestReportBase
VAR_INPUT
END_VAR
VAR_OUTPUT
END_VAR
VAR
END_VAR

(******************************************************************************
Baustein: FB_TestReportBase.BuildFile
Spezifikation: doc/Spezifikation.pdf, Kap. x.y.z
-------------------------------------------------------------------------------
erstellt:
von:
Geändert:
von:
-------------------------------------------------------------------------------
Beschreibung
Diese Methode muss vom ableitenden Baustein überschrieben werden und
wird von der Basisklasse aus aufgerufen wenn der Report erstellt werden
soll.

-------------------------------------------------------------------------------
Input
-

Output
-
******************************************************************************)
METHOD PROTECTED BuildFile : ERetCode_t
VAR_INPUT
	i_u32Line : UDINT;
END_VAR

	BuildFile := ERetCode_t.eRetBusy;

	CASE i_u32Line OF

	0: addString('Test Report ');
	
	1: addString('++++++++++++++++++++++++++++++++++++++++++++++++++');

	2: addString('Ergebnis');
	
	3: addString('++++++++++++++++++++++++++++++++++++++++++++++++++');
	
	4: BuildFile := ERetCode_t.eRetDone;

	END_CASE;
END_METHOD

(******************************************************************************
Baustein: FB_TestReportBase.getFileName
Spezifikation: doc/Spezifikation.pdf, Kap. x.y.z
-------------------------------------------------------------------------------
erstellt:
von:
Geändert:
von:
-------------------------------------------------------------------------------
Beschreibung
Diese Methode muss vom ableitenden Baustein überschrieben werden und
wird von der Basisklasse aus aufgerufen wenn der Report erstellt werden
soll.

-------------------------------------------------------------------------------
Input
-

Output
-
******************************************************************************)
METHOD PROTECTED getFileName : ERetCode_t
VAR_INPUT
	i_pFileName : NameHandle_t;
	i_pPath		: PathHandle_t;
END_VAR

	i_pFileName^ := 'Export.txt';
	i_pPath^ 	 := 'C:\Users\Administrator\Desktop\';
END_METHOD

END_FUNCTION_BLOCK
